(* IEC 61131-3 sources: AXOpen/src/io/ctrl/src/AxoIoComponent/TypesStructuresAndEnums, 9 files *)

(* ---- ComponentState.st ---- *)
NAMESPACE AXOpen.Io
    TYPE ComponentState : UINT (
        Good                    :=	UINT#0, //	No problems detected.
        Disabled                :=	UINT#1, //	The hardware component is disabled.
        MaintenanceRequired     :=	UINT#2, //	Maintenance required.
        MaintenanceDemanded     :=	UINT#3, //	Maintenance demanded.
        Error                   :=	UINT#4, //	Error.
        NotAccessible           :=	UINT#5, //	Status unknown or error in higher-level hardware component.
        Unknown                 :=	UINT#6, //	Default value for components that do not return diagnostic events.
        IONotAvailable          :=	UINT#7  //	Inputs/outputs are not available.
                    ) := Unknown;
    END_TYPE
END_NAMESPACE

(* ---- OperatingState.st ---- *)
NAMESPACE AXOpen.Io
    TYPE OperatingState : UINT (
        Unknown                     :=  UINT#255,
        NotSupported                :=	UINT#0,     //	Not Supported; for I/O modules OperatingState always has this value.
        StopFirmwareUpdate          :=	UINT#1,     //	STOP; firmware update.
        StopMemoryReset             :=	UINT#2,     //	STOP; memory reset.
        StopSelfStart               :=	UINT#3,     //	STOP; self start.
        Stop                        :=	UINT#4,     //	STOP.
        MemoryReset                 :=	UINT#5,     //	Memory reset.
        Startup                     :=	UINT#6,     //	STARTUP.
        Run                         :=	UINT#8,     //	RUN.
        RunRedundant                :=	UINT#9,     //	RUN-REDUNDANT.
        Hold                        :=	UINT#10,    //	HOLD.
        Defect                      :=	UINT#13,    //	DEFECT (can only be seen in diagnostic buffer entries).
        DeEnergized                 :=	UINT#15,    //	De-energized (can only be seen in diagnostic buffer entries).
        ConfigurationInRun          :=	UINT#16,    //	Configuration in Run (CiR).
        StopWithoutOutputDisable    :=	UINT#17,    //	STOP without output disable.
        RunWithOutputDisable        :=	UINT#18,    //	RUN with output disable.
        PgmTest                     :=	UINT#19,    //	PgmTest.
        PrimaryRunBackupTest        :=	UINT#20,    //	RunPgmTest (state of primary PLC when the backup PLC is in test mode).
        PrimarySyncup               :=	UINT#21,    //	RUN-SYNCUP (only primary PLC in SYNCUP system state).
        BackupSyncup                :=	UINT#22,    //	SYNCUP (only backup PLC in SYNCUP system state)
        PartnerPlcStateUnknown      :=	UINT#31,    //	State of partner PLC unknown (for example when the partner PLC is not available).
        StopSystemState             :=	UINT#33,    //	STOP system state
        StartupSystemState          :=	UINT#35,    //	STARTUP system state
        RunSoloSystemState          :=	UINT#37,    //	RUN-SOLO system state
        SyncupSystemState           :=	UINT#38,    //	SYNCUP system state
        RunRedundantSystemState     :=	UINT#40    //	RUN-REDUNDANT system state
                    ) := Unknown;
    END_TYPE
END_NAMESPACE

(* ---- ReplacementState.st ---- *)
NAMESPACE AXOpen.Io
    TYPE ReplacementState : UINT (
        Unknown         :=	UINT#255,
        OK              :=	UINT#0, //	The correct element exists.
        Substitute      :=	UINT#1, //	The element was replaced by a compatible element.
        Incompatible    :=	UINT#2, //	The element was replaced by an incompatible element (is reachable, but not ready for operation).
        Missing         :=	UINT#3 //	The element does not exist.
            ) := Unknown;
    END_TYPE
END_NAMESPACE

(* ---- ComponentStateDetail.st ---- *)
NAMESPACE AXOpen.Io
    {S7.extern=ReadWrite}
    CLASS ComponentStateDetail
		VAR PUBLIC
            {#ix-attr:[Container(Layout.Wrap)]}
            {#ix-attr:[Group(GroupLayout.GroupBox)]}
            {#ix-set:AttributeName = "<#Hardware component state#>"}
            HardwareComponentState  :   HardwareComponentState;  //	Represents detailed state information about the hardware component.
            {#ix-attr:[Container(Layout.Wrap)]}
            {#ix-attr:[Group(GroupLayout.GroupBox)]}
            {#ix-set:AttributeName = "<#PlcState#>"}
            PlcState                :	PlcState;                //	Represents detailed state information about the PLC.
        END_VAR
    END_CLASS
END_NAMESPACE

(* ---- DiagnosticDetails .st ---- *)
NAMESPACE AXOpen.Io
    {S7.extern=ReadWrite}
    CLASS DiagnosticDetails
        VAR PUBLIC
            {#ix-attr:[Container(Layout.Wrap)]}
            {#ix-attr:[Group(GroupLayout.GroupBox)]}
            {#ix-set:AttributeName = "<#Component state detail#>"}
            ComponentStateDetail    :	ComponentStateDetail;	//  Represents detailed state information about the hardware component and the PLC.
            {#ix-attr:[Container(Layout.Wrap)]}
            {#ix-attr:[Group(GroupLayout.GroupBox)]}
            {#ix-set:AttributeName = "<#Component state#>"}
            ComponentState          :	ComponentState;	        //  State of the component.
            {#ix-attr:[Container(Layout.Wrap)]}
            {#ix-attr:[Group(GroupLayout.GroupBox)]}
            {#ix-set:AttributeName = "<#IO state#>"}
            IOState                 :	IOState;	            //  State of the inputs and outputs of the component.
            {#ix-attr:[Container(Layout.Wrap)]}
            {#ix-attr:[Group(GroupLayout.GroupBox)]}
            {#ix-set:AttributeName = "<#Operating state#>"}
            OperatingState           :	OperatingState;	        //  Operating state of the PLC.
        END_VAR
    END_CLASS
END_NAMESPACE

(* ---- DiagnosticDetails.st ---- *)
NAMESPACE AXOpen.Io
    {S7.extern=ReadWrite}
    CLASS DiagnosticDetails
        VAR PUBLIC
            {#ix-attr:[Container(Layout.Wrap)]}
            {#ix-attr:[Group(GroupLayout.GroupBox)]}
            {#ix-set:AttributeName = "<#Component state detail#>"}
            ComponentStateDetail    :	ComponentStateDetail;	//  Represents detailed state information about the hardware component and the PLC.
            {#ix-attr:[Container(Layout.Wrap)]}
            {#ix-attr:[Group(GroupLayout.GroupBox)]}
            {#ix-set:AttributeName = "<#Component state#>"}
            ComponentState          :	ComponentState;	        //  State of the component.
            {#ix-attr:[Container(Layout.Wrap)]}
            {#ix-attr:[Group(GroupLayout.GroupBox)]}
            {#ix-set:AttributeName = "<#IO state#>"}
            IOState                 :	IOState;	            //  State of the inputs and outputs of the component.
            {#ix-attr:[Container(Layout.Wrap)]}
            {#ix-attr:[Group(GroupLayout.GroupBox)]}
            {#ix-set:AttributeName = "<#Operating state#>"}
            OperatingState           :	OperatingState;	        //  Operating state of the PLC.
        END_VAR
    END_CLASS
END_NAMESPACE

(* ---- HardwareComponentState.st ---- *)
NAMESPACE AXOpen.Io
    {S7.extern=ReadWrite}
    CLASS HardwareComponentState
	VAR PUBLIC
            {#ix-attr:[Container(Layout.Stack)]}
            NoAdditionalInformation     :	BOOL;	//  No additional information available.
            TransferNotPermitted        :	BOOL;	//  Transfer not permitted.
            DiagnosticsAvailable        :	BOOL;	//  At least one qualified diagnostics is available.
            MaintenanceRequired         :	BOOL;	//  Maintenance required for at least one channel or the component.
            MaintenanceDemanded         :	BOOL;	//  Maintenance demanded for at least one channel or the component.
            Error                       :	BOOL;	//  Error in at least one channel or the component.
            ComponentAvailability	    :   ComponentAvailability;
            ReplacementState	        :   ReplacementState;
        END_VAR
    END_CLASS
END_NAMESPACE

(* ---- IOState.st ---- *)
NAMESPACE AXOpen.Io
    {S7.extern=ReadWrite}
    CLASS IOState
        VAR PUBLIC
            {#ix-attr:[Container(Layout.Stack)]}
            Good                    :	BOOL;   //	No problems detected.
            Disabled                :	BOOL;   //	The hardware component is disabled.
            MaintenanceRequired     :	BOOL;   //	Maintenance required.
            MaintenanceDemanded     :	BOOL;   //	Maintenance demanded.
            Error                   :	BOOL;   //	Error.
            NotAccessible           :	BOOL;   //	Hardware component not reachable; hardware component cannot be accessed.
            DiagnosticsAvailable    :	BOOL;   //	At least one qualified diagnostics is available.
            IODataNotAvailable      :	BOOL;   //	I/O data not available.
            NetworkError            :	BOOL;   //	Network error.
            HardwareError           :	BOOL;   //	Hardware error.
        END_VAR
    END_CLASS
END_NAMESPACE

(* ---- SubordinateDiagnosticDetails.st ---- *)
NAMESPACE AXOpen.Io
    {S7.extern=ReadWrite}
    CLASS SubordinateDiagnosticDetails
        VAR PUBLIC
            {#ix-attr:[Container(Layout.Wrap)]}
            {#ix-set:AttributeName = "<#Subordinate state#>"}
            SubordinateState          :	ComponentState;
            {#ix-set:AttributeName = "<#Subordinate IO state#>"}
            SubordinateIOState                 :	IOState;
            {#ix-set:AttributeName = "<#Operating DiagnosticsEnabled#>"}
            DiagnosticsEnabled           :	BOOL;
        END_VAR
    END_CLASS
END_NAMESPACE
